KUKA KRL program: service1.src, service1.dat

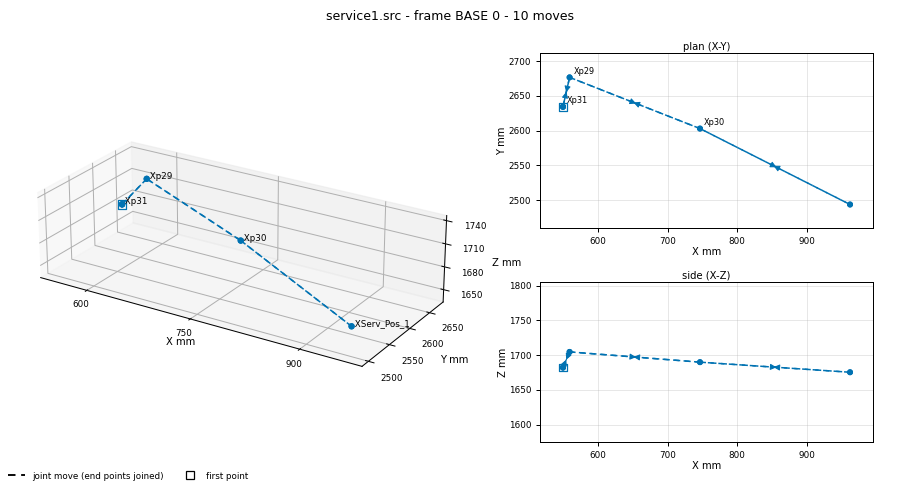
[picture p0: tool path of service1.src in frame BASE 0, 10 of 11 moves have a stored position in this frame; points joined in program order, loops and branches not executed]
--- service1.src ---
&ACCESS RVP1
&REL 125
&COMMENT MANTENIMIENTO
DEF SERVICE1( )
;================================================
; MODELO   : C-520
; IE GRUPO : 5J
; ESTACION : 85
; ROBOT    : 85R02
; FUNCTION : MAINTENANCE PROGRAM
;================================================
;FOLD INI
;FOLD BASISTECH INI
GLOBAL INTERRUPT DECL 3 WHEN $STOPMESS==TRUE DO IR_STOPM ( )
INTERRUPT ON 3
BAS (#INITMOV,0 )
;ENDFOLD (BASISTECH INI)
;FOLD SPOTTECH INI
;USERSPOT(#INIT)
;ENDFOLD (SPOTTECH INI)
;FOLD GRIPPERTECH INI
USER_GRP(0,DUMMY,DUMMY,GDEFAULT)
;ENDFOLD (GRIPPERTECH INI)
;FOLD USER INI
;Make your modifications here
;base_corr_on=true
;base_corr.a=-45
;ENDFOLD (USER INI)
;ENDFOLD (INI)

;FOLD PTP home Vel=100 % H;%{PE}%R 5.6.13,%MKUKATPBASIS,%CMOVE,%VPTP,%P 1:PTP, 2:home, 3:, 5:100, 7:H
$BWDSTART=FALSE
PDAT_ACT=PH
FDAT_ACT=Fhome
BAS(#PTP_PARAMS,100)
$H_POS=XHOME
PTP Xhome
;ENDFOLD




;FOLD PTP p31 Vel=75 % H Tool[0] Base[0];%{PE}%R 5.6.13,%MKUKATPBASIS,%CMOVE,%VPTP,%P 1:PTP, 2:p31, 3:, 5:75, 7:H
$BWDSTART=FALSE
PDAT_ACT=PH
FDAT_ACT=Fp31
BAS(#PTP_PARAMS,75)
PTP Xp31
;ENDFOLD
;FOLD PTP p27 Vel=75 % H Tool[0] Base[0];%{PE}%R 5.6.13,%MKUKATPBASIS,%CMOVE,%VPTP,%P 1:PTP, 2:p27, 3:, 5:75, 7:H
$BWDSTART=FALSE
PDAT_ACT=PH
FDAT_ACT=Fp27
BAS(#PTP_PARAMS,75)
PTP Xp27
;ENDFOLD
;FOLD PTP p29 Vel=75 % H Tool[0] Base[0];%{PE}%R 5.6.13,%MKUKATPBASIS,%CMOVE,%VPTP,%P 1:PTP, 2:p29, 3:, 5:75, 7:H
$BWDSTART=FALSE
PDAT_ACT=PH
FDAT_ACT=Fp29
BAS(#PTP_PARAMS,75)
PTP Xp29
;ENDFOLD
;FOLD PTP p30 Vel=75 % H Tool[0] Base[0];%{PE}%R 5.6.13,%MKUKATPBASIS,%CMOVE,%VPTP,%P 1:PTP, 2:p30, 3:, 5:75, 7:H
$BWDSTART=FALSE
PDAT_ACT=PH
FDAT_ACT=Fp30
BAS(#PTP_PARAMS,75)
PTP Xp30
;ENDFOLD
;FOLD PTP Serv_Pos_1 Vel=75 % H Tool[0] Base[0];%{PE}%R 5.6.13,%MKUKATPBASIS,%CMOVE,%VPTP,%P 1:PTP, 2:Serv_Pos_1, 3:, 5:75, 7:H
$BWDSTART=FALSE
PDAT_ACT=PH
FDAT_ACT=FServ_Pos_1
BAS(#PTP_PARAMS,75)
PTP XServ_Pos_1
;ENDFOLD

; Maintenance position
O_SERVP=TRUE

if false then
serv2galga()
endif

if false then
serv2foto()
endif

;Wait return to home
WAIT FOR I_RETHP == TRUE

;FOLD PTP serv_pos_1 Vel=75 % H Tool[0] Base[0];%{PE}%R 5.6.13,%MKUKATPBASIS,%CMOVE,%VPTP,%P 1:PTP, 2:serv_pos_1, 3:, 5:75, 7:H
$BWDSTART=FALSE
PDAT_ACT=PH
FDAT_ACT=Fserv_pos_1
BAS(#PTP_PARAMS,75)
PTP Xserv_pos_1
;ENDFOLD
;FOLD PTP p30 Vel=75 % H Tool[0] Base[0];%{PE}%R 5.6.13,%MKUKATPBASIS,%CMOVE,%VPTP,%P 1:PTP, 2:p30, 3:, 5:75, 7:H
$BWDSTART=FALSE
PDAT_ACT=PH
FDAT_ACT=Fp30
BAS(#PTP_PARAMS,75)
PTP Xp30
;ENDFOLD
;FOLD PTP p29 Vel=75 % H Tool[0] Base[0];%{PE}%R 5.6.13,%MKUKATPBASIS,%CMOVE,%VPTP,%P 1:PTP, 2:p29, 3:, 5:75, 7:H
$BWDSTART=FALSE
PDAT_ACT=PH
FDAT_ACT=Fp29
BAS(#PTP_PARAMS,75)
PTP Xp29
;ENDFOLD
;FOLD PTP p27 Vel=75 % H Tool[0] Base[0];%{PE}%R 5.6.13,%MKUKATPBASIS,%CMOVE,%VPTP,%P 1:PTP, 2:p27, 3:, 5:75, 7:H
$BWDSTART=FALSE
PDAT_ACT=PH
FDAT_ACT=Fp27
BAS(#PTP_PARAMS,75)
PTP Xp27
;ENDFOLD
;FOLD PTP p31 Vel=75 % H Tool[0] Base[0];%{PE}%R 5.6.13,%MKUKATPBASIS,%CMOVE,%VPTP,%P 1:PTP, 2:p31, 3:, 5:75, 7:H
$BWDSTART=FALSE
PDAT_ACT=PH
FDAT_ACT=Fp31
BAS(#PTP_PARAMS,75)
PTP Xp31
;ENDFOLD
O_SERVP=FALSE

END

--- service1.dat ---
&ACCESS RVP1
&REL 125
&COMMENT MANTENIMIENTO
DEFDAT  SERVICE1
;FOLD EXTERNAL DECLARATIONS;%{PE}%V3.2.0,%MKUKATPBASIS,%CEXT,%VCOMMON,%P
;FOLD GRIPPERTECH EXT
EXT  H50 (INT  :IN,INT  :IN,INT  :IN,GRP_TYP  :IN )
;ENDFOLD (GRIPPERTECH EXT)
;FOLD SPOTTECH EXT
EXT  USERSPOT (S_COMMAND  :IN,SPOT_TYPE  :IN )
;ENDFOLD (SPOTTECH EXT)
;FOLD BAS EXT;%{PE}%V3.2.0,%MKUKATPBASIS,%CEXT,%VEXT,%P
EXT  BAS (BAS_COMMAND  :IN,REAL  :IN )
DECL INT SUCCESS
;ENDFOLD
;FOLD USER EXT;%{E}%V3.2.0,%MKUKATPUSER,%CEXT,%VEXT,%P
;Make here your modifications
;ENDFOLD
;ENDFOLD
;FOLD USER EXT;%{}%V2.2.2,%MKUKATPUSER,%CEXT,%VEXT,%P
;Make here your modifications
DECL BOOL TIPKONTROLE
DECL INT ANSWER
DECL INT WAITTIME=1000
;ENDFOLD
;ENDFOLD
DECL INT I

;******************************
;*     E6POS Declarations     *
;******************************

DECL E6POS XP10={X 1528.24902,Y -682.445679,Z 1907.06006,A 2.01388311,B -48.187439,C 158.723099,S 2,T 42,E1 0.0,E2 0.0,E3 0.0,E4 0.0,E5 0.0,E6 0.0}
DECL E6POS XSERV_POS_1={X 962.371399,Y 2493.73804,Z 1675.50305,A -175.466293,B 44.8439293,C -178.865295,S 2,T 35,E1 0.0,E2 0.0,E3 0.0,E4 0.0,E5 0.0,E6 0.0}
DECL E6POS XP20={X 1962.03003,Y 188.434097,Z 1762.45703,A 18.2867107,B 83.2636337,C -1.26252997,S 6,T 51,E1 0.0,E2 0.0,E3 0.0,E4 0.0,E5 0.0,E6 0.0}

;******************************
;*      FDAT Declarations     *
;******************************

DECL FDAT FP10={TOOL_NO 14,BASE_NO 0,IPO_FRAME #BASE,TQ_STATE FALSE}
DECL FDAT FSERV_POS_1={TOOL_NO 0,BASE_NO 0,IPO_FRAME #BASE,TQ_STATE FALSE}
DECL FDAT FP20={TOOL_NO 14,BASE_NO 0,IPO_FRAME #BASE,TQ_STATE FALSE}

;******************************
;*  PDAT & LDAT Declarations  *
;******************************

DECL PDAT PH={VEL 100.0,ACC 100.0,APO_DIST 100.0,APO_MODE #CPTP}

DECL SPOT_SUGG_T LAST_SPOT={GUN[] "1                       ",RETR_CMD[] "#OPN                    ",CHOISE[] "#FIRST                  ",CLO_TM[] "0                       ",PGNO1[] "1                       ",PRESS1[] "0                       ",PGNO2[] "1                       ",PRESS2[] "0                       ",SPOT_PARAMS[] "SDAT0                   "}
DECL BASIS_SUGG_T LAST_BASIS={POINT1[] "p31                     ",POINT2[] "p31                     ",CP_PARAMS[] "CPDAT0                  ",PTP_PARAMS[] "H                       ",CONT[] "                        ",CP_VEL[] "2                       ",PTP_VEL[] "100                     ",SYNC_PARAMS[] "SYNCDAT                 ",SPL_NAME[] "S0                      "}
DECL INT LAST_XP_POINT=0
DECL E6POS XP1={X 1335.83801,Y -1478.72205,Z 1732.87097,A -27.0469608,B -54.993309,C 160.553802,S 2,T 42,E1 0.0,E2 0.0,E3 0.0,E4 0.0,E5 0.0,E6 0.0}
DECL FDAT FP1={TOOL_NO 14,BASE_NO 0,IPO_FRAME #BASE,POINT2[] " ",TQ_STATE FALSE}
DECL E6POS XP2={X 1335.83801,Y -1478.72205,Z 1732.87097,A -27.0469608,B -54.993309,C 160.553802,S 2,T 42,E1 0.0,E2 0.0,E3 0.0,E4 0.0,E5 0.0,E6 0.0}
DECL FDAT FP2={TOOL_NO 14,BASE_NO 0,IPO_FRAME #BASE,POINT2[] " ",TQ_STATE FALSE}
DECL LDAT LCPDAT6={VEL 2.0,ACC 100.0,APO_DIST 100.0,APO_FAC 50.0,ORI_TYP #VAR,CIRC_TYP #BASE,JERK_FAC 50.0,EXAX_IGN 0}
DECL E6POS XP3={X 1962.03296,Y 188.453506,Z 1762.45496,A 18.2838898,B 83.2638702,C -1.26579797,S 6,T 50,E1 0.0,E2 0.0,E3 0.0,E4 0.0,E5 0.0,E6 0.0}
DECL FDAT FP3={TOOL_NO 14,BASE_NO 0,IPO_FRAME #BASE,POINT2[] " ",TQ_STATE FALSE}
DECL E6POS XP4={X 2060.22095,Y -757.729919,Z 331.827606,A 72.5727005,B -0.352961212,C 118.131203,S 5,T 23,E1 0.0,E2 0.0,E3 0.0,E4 0.0,E5 0.0,E6 0.0}
DECL FDAT FP4={TOOL_NO 14,BASE_NO 0,IPO_FRAME #BASE,POINT2[] " ",TQ_STATE FALSE}
DECL E6POS XPOSICION_SERVICIO={X 2378.94897,Y -515.166504,Z 615.737427,A 139.647095,B -1.39994705,C 79.0117493,S 1,T 7,E1 0.0,E2 0.0,E3 0.0,E4 0.0,E5 0.0,E6 0.0}
DECL FDAT Fposicion_servicio={TOOL_NO 14,BASE_NO 0,IPO_FRAME #BASE,POINT2[] " ",TQ_STATE FALSE}
DECL E6POS XP6={X 648.720886,Y -752.985718,Z 867.136902,A -112.871597,B -3.13271499,C -172.899094,S 6,T 26,E1 0.0,E2 0.0,E3 0.0,E4 0.0,E5 0.0,E6 0.0}
DECL FDAT Fp6={TOOL_NO 14,BASE_NO 0,IPO_FRAME #BASE,POINT2[] " ",TQ_STATE FALSE}
DECL E6POS Xp7={X 735.259827,Y -846.376282,Z -50.7595787,A 36.4931488,B 2.33025098,C -7.71590185,S 6,T 26,E1 0.0,E2 0.0,E3 0.0,E4 0.0,E5 0.0,E6 0.0}
DECL FDAT Fp7={TOOL_NO 1,BASE_NO 0,IPO_FRAME #BASE,POINT2[] " ",TQ_STATE FALSE}
DECL E6POS Xp8={X 481.643494,Y -1154.31702,Z -148.6595,A 30.6545601,B 3.87480402,C -9.08418941,S 6,T 26,E1 0.0,E2 0.0,E3 0.0,E4 0.0,E5 0.0,E6 0.0}
DECL FDAT Fp8={TOOL_NO 1,BASE_NO 0,IPO_FRAME #BASE,POINT2[] " ",TQ_STATE FALSE}
DECL E6POS Xp9={X 17.5958195,Y -1360.61597,Z -301.022308,A 23.6130409,B 6.36468601,C -9.25088882,S 6,T 26,E1 0.0,E2 0.0,E3 0.0,E4 0.0,E5 0.0,E6 0.0}
DECL FDAT Fp9={TOOL_NO 1,BASE_NO 0,IPO_FRAME #BASE,POINT2[] " ",TQ_STATE FALSE}
DECL E6POS Xp11={X 735.259827,Y -846.376282,Z -50.7595787,A 36.4931488,B 2.33025098,C -7.71590185,S 6,T 26,E1 0.0,E2 0.0,E3 0.0,E4 0.0,E5 0.0,E6 0.0}
DECL FDAT Fp11={TOOL_NO 1,BASE_NO 0,IPO_FRAME #BASE,POINT2[] " ",TQ_STATE FALSE}
DECL E6POS Xp12={X 481.643494,Y -1154.31702,Z -148.6595,A 30.6545601,B 3.87480402,C -9.08418941,S 6,T 26,E1 0.0,E2 0.0,E3 0.0,E4 0.0,E5 0.0,E6 0.0}
DECL FDAT Fp12={TOOL_NO 1,BASE_NO 0,IPO_FRAME #BASE,POINT2[] " ",TQ_STATE FALSE}
DECL E6POS Xp13={X 17.5958195,Y -1360.61597,Z -301.022308,A 23.6130409,B 6.36468601,C -9.25088882,S 6,T 26,E1 0.0,E2 0.0,E3 0.0,E4 0.0,E5 0.0,E6 0.0}
DECL FDAT Fp13={TOOL_NO 1,BASE_NO 0,IPO_FRAME #BASE,POINT2[] " ",TQ_STATE FALSE}
DECL E6POS Xp14={X 735.259827,Y -846.376282,Z -50.7595787,A 36.4931488,B 2.33025098,C -7.71590185,S 6,T 26,E1 0.0,E2 0.0,E3 0.0,E4 0.0,E5 0.0,E6 0.0}
DECL FDAT Fp14={TOOL_NO 1,BASE_NO 0,IPO_FRAME #BASE,POINT2[] " ",TQ_STATE FALSE}
DECL E6POS Xp15={X 481.643494,Y -1154.31702,Z -148.6595,A 30.6545601,B 3.87480402,C -9.08418941,S 6,T 26,E1 0.0,E2 0.0,E3 0.0,E4 0.0,E5 0.0,E6 0.0}
DECL FDAT Fp15={TOOL_NO 1,BASE_NO 0,IPO_FRAME #BASE,POINT2[] " ",TQ_STATE FALSE}
DECL E6POS Xp16={X 17.5958195,Y -1360.61597,Z -301.022308,A 23.6130409,B 6.36468601,C -9.25088882,S 6,T 26,E1 0.0,E2 0.0,E3 0.0,E4 0.0,E5 0.0,E6 0.0}
DECL FDAT Fp16={TOOL_NO 1,BASE_NO 0,IPO_FRAME #BASE,POINT2[] " ",TQ_STATE FALSE}
DECL E6POS Xp17={X 1.47015905,Y -1176.46594,Z -326.900909,A 24.0927391,B 2.20976591,C -0.817254126,S 6,T 26,E1 0.0,E2 0.0,E3 0.0,E4 0.0,E5 0.0,E6 0.0}
DECL FDAT Fp17={TOOL_NO 1,BASE_NO 0,IPO_FRAME #BASE,POINT2[] " ",TQ_STATE FALSE}
DECL E6POS XP18={X 1254.51501,Y -344.527496,Z 2.55625296,A 63.4769592,B 0.486176193,C -13.7634096,S 6,T 26,E1 0.0,E2 0.0,E3 0.0,E4 0.0,E5 0.0,E6 0.0}
DECL FDAT Fp18={TOOL_NO 1,BASE_NO 0,IPO_FRAME #BASE,POINT2[] " ",TQ_STATE FALSE}
DECL E6POS XP19={X 481.645599,Y -1154.23706,Z -148.684402,A 30.6538391,B 3.8741889,C -9.08234215,S 6,T 26,E1 0.0,E2 0.0,E3 0.0,E4 0.0,E5 0.0,E6 0.0}
DECL FDAT Fp19={TOOL_NO 1,BASE_NO 0,IPO_FRAME #BASE,POINT2[] " ",TQ_STATE FALSE}
DECL E6POS XP21={X 17.6284695,Y -1360.54199,Z -301.040405,A 23.6120491,B 6.36356592,C -9.2495842,S 6,T 26,E1 0.0,E2 0.0,E3 0.0,E4 0.0,E5 0.0,E6 0.0}
DECL FDAT Fp21={TOOL_NO 1,BASE_NO 0,IPO_FRAME #BASE,POINT2[] " ",TQ_STATE FALSE}
DECL E6POS XP22={X 481.643707,Y -1154.25903,Z -148.675705,A 30.6532707,B 3.87440109,C -9.08279896,S 6,T 26,E1 0.0,E2 0.0,E3 0.0,E4 0.0,E5 0.0,E6 0.0}
DECL FDAT Fp22={TOOL_NO 1,BASE_NO 0,IPO_FRAME #BASE,POINT2[] " ",TQ_STATE FALSE}
DECL E6POS XP23={X -908.508301,Y -1450.92297,Z -250.134399,A -2.65489292,B 0.133399099,C 0.548784316,S 6,T 26,E1 0.0,E2 0.0,E3 0.0,E4 0.0,E5 0.0,E6 0.0}
DECL FDAT Fp23={TOOL_NO 1,BASE_NO 0,IPO_FRAME #BASE,POINT2[] " ",TQ_STATE FALSE}
DECL E6POS XP24={X -957.974426,Y -1455.21802,Z 675.247925,A -152.189499,B 2.96034288,C -178.895294,S 6,T 26,E1 0.0,E2 0.0,E3 0.0,E4 0.0,E5 0.0,E6 0.0}
DECL FDAT Fp24={TOOL_NO 14,BASE_NO 0,IPO_FRAME #BASE,POINT2[] " ",TQ_STATE FALSE}
DECL E6POS XP25={X 1254.51501,Y -344.527496,Z 2.55625296,A 63.4769592,B 0.486176193,C -13.7634096,S 6,T 26,E1 0.0,E2 0.0,E3 0.0,E4 0.0,E5 0.0,E6 0.0}
DECL FDAT Fp25={TOOL_NO 1,BASE_NO 0,IPO_FRAME #BASE,POINT2[] " ",TQ_STATE FALSE}
DECL E6POS XP26={X 1025.29395,Y 45.5070381,Z -7.78524017,A 66.922142,B 0.952350318,C -4.80453396,S 6,T 26,E1 0.0,E2 0.0,E3 0.0,E4 0.0,E5 0.0,E6 0.0}
DECL FDAT Fp26={TOOL_NO 1,BASE_NO 0,IPO_FRAME #BASE,POINT2[] " ",TQ_STATE FALSE}
DECL E6POS XP27={X 549.68811,Y 2634.30103,Z 1682.375,A -89.872551,B 18.4036407,C -135.711502,S 2,T 3,E1 0.0,E2 0.0,E3 0.0,E4 0.0,E5 0.0,E6 0.0}
DECL FDAT Fp27={TOOL_NO 0,BASE_NO 0,IPO_FRAME #BASE,POINT2[] " ",TQ_STATE FALSE}
DECL E6POS XP28={X 686.024597,Y 2590.84912,Z 1678.09399,A -133.558197,B 40.0909996,C -155.806503,S 2,T 35,E1 0.0,E2 0.0,E3 0.0,E4 0.0,E5 0.0,E6 0.0}
DECL FDAT Fp28={TOOL_NO 0,BASE_NO 0,IPO_FRAME #BASE,POINT2[] " ",TQ_STATE FALSE}
DECL E6POS XP29={X 559.20813,Y 2676.47803,Z 1704.76099,A -133.993896,B 53.4526291,C -167.733902,S 2,T 35,E1 0.0,E2 0.0,E3 0.0,E4 0.0,E5 0.0,E6 0.0}
DECL FDAT Fp29={TOOL_NO 0,BASE_NO 0,IPO_FRAME #BASE,POINT2[] " ",TQ_STATE FALSE}
DECL E6POS XP30={X 746.671387,Y 2602.89502,Z 1689.99597,A -169.726593,B 49.4236908,C 173.351501,S 2,T 35,E1 0.0,E2 0.0,E3 0.0,E4 0.0,E5 0.0,E6 0.0}
DECL FDAT Fp30={TOOL_NO 0,BASE_NO 0,IPO_FRAME #BASE,POINT2[] " ",TQ_STATE FALSE}
DECL E6POS XP31={X 549.688171,Y 2634.302,Z 1682.37402,A -31.6532898,B -34.9410095,C -145.953201,S 2,T 3,E1 0.0,E2 0.0,E3 0.0,E4 0.0,E5 0.0,E6 0.0}
DECL FDAT Fp31={TOOL_NO 0,BASE_NO 0,IPO_FRAME #BASE,POINT2[] " ",TQ_STATE FALSE}
ENDDAT
